ABB RobotStudio station: Assignment2_task#2_20200910-153317.rsstn

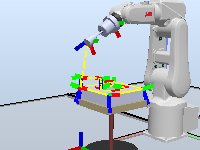
Station Assignment2_task#2 (saved by RobotStudio 20.1.9014.1)
Controller Controller3, task T_ROB1: task frame (RAPID world) sits at (100, 100, 0) mm in the station
Controller Controller3
  mechanical unit ROB_1: IRB120_3_58__01, 6 joints, base frame (0, 0, 0) mm
Layout (positions relative to the parent item):
  - IRB120_3_58__01 [mechanism, from Robots\IRB120_3_58_G_01.rslib] at (100, 100, 0) mm; joint values [0, 0, 0, 0, 0.5236, 0] (rad or m)
  - AssemblySpindleSide [part] at (447.83, 171.64, 630.14) mm, rotated rx -90 ry 60 rz 180 deg
  - Task2_Part [part] at (570, 0, 250) mm, rotated rx 90 ry 0 rz 90 deg
  - Table [part] at (15, -15, 220) mm
  - LegBase [part] at (-100, 100, 0) mm
  - LegSupport [part] at (-100, 100, 0) mm
Attachment: AssemblySpindleSide is attached to IRB120_3_58__01 / Link6
Attachment: LegSupport is attached to Table
Attachment: LegBase is attached to LegSupport
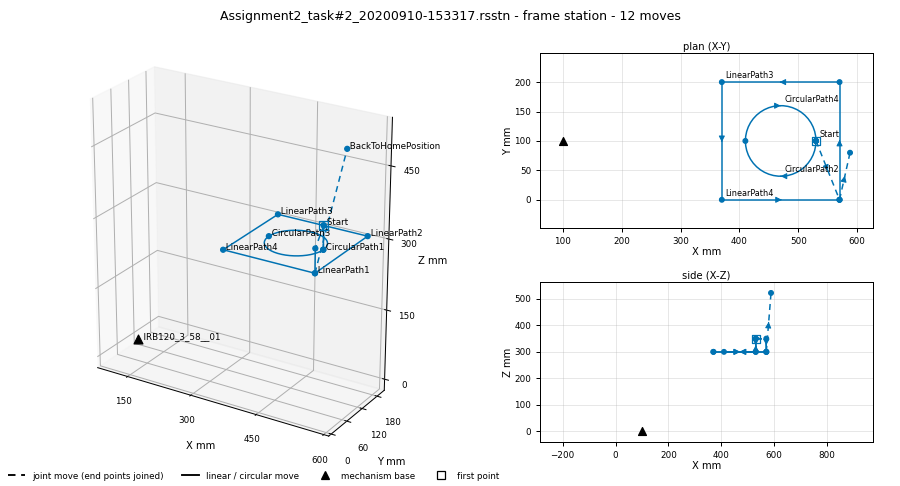
[picture p0: tool path of Assignment2_task#2_20200910-153317.rsstn in frame station, 12 of 12 moves have a stored position in this frame; points joined in program order, loops and branches not executed]
Targets, tools, work objects and paths stored in the station, written as RAPID:
! task T_ROB1
MODULE CalibData
  TASK PERS tooldata Tooldata_1:=[TRUE,[[0,-20.001,142.61],[1,0,0,0]],[1,[0,0,1],[1,0,0,0],0,0,0]];
  TASK PERS wobjdata task2:=[FALSE,TRUE,"",[[470,-100,0],[0.707106781,0,0,0.707106781]],[[0,0,0],[1,0,0,0]]];
  TASK PERS wobjdata LegBase:=[FALSE,TRUE,"",[[470,-100,10],[1,0,0,0]],[[0,0,0],[1,0,0,0]]];
ENDMODULE

! task T_ROB1
MODULE Module1
  CONST robtarget CircularPath1:=[[100,40,300],[0,0,0.984807753,0.173648179],[0,0,-1,0],[9E+09,9E+09,9E+09,9E+09,9E+09,9E+09]];
  CONST robtarget CircularPath2:=[[40,100,300],[0.122787804,0.69636424,0.69636424,0.122787804],[-1,0,-1,0],[9E+09,9E+09,9E+09,9E+09,9E+09,9E+09]];
  CONST robtarget CircularPath3:=[[100,160,300],[0.130526193,0.991444861,0,0],[0,0,0,0],[9E+09,9E+09,9E+09,9E+09,9E+09,9E+09]];
  CONST robtarget CircularPath4:=[[160,100,300],[0.122787804,0.69636424,-0.69636424,-0.122787804],[0,-1,2,0],[9E+09,9E+09,9E+09,9E+09,9E+09,9E+09]];
  CONST robtarget CircularPath5:=[[100,40,300],[0,0,0.984807753,0.173648178],[0,-1,2,0],[9E+09,9E+09,9E+09,9E+09,9E+09,9E+09]];
  CONST robtarget Start:=[[100,40,350],[0,0,1,0],[0,0,-1,0],[9E+09,9E+09,9E+09,9E+09,9E+09,9E+09]];
  CONST robtarget lift:=[[100,40,350],[0,0,1,0],[0,0,3,0],[9E+09,9E+09,9E+09,9E+09,9E+09,9E+09]];
  CONST robtarget Start2:=[[0,0,350],[0,1,0,0],[-1,0,0,0],[9E+09,9E+09,9E+09,9E+09,9E+09,9E+09]];
  CONST robtarget Lift2:=[[0,0,350],[0,-0.707106781,0.707106781,0],[-1,0,-3,0],[9E+09,9E+09,9E+09,9E+09,9E+09,9E+09]];
  CONST robtarget BackToHomePosition:=[[17.857711906,79.999,512.695],[0.5,0,0.866025404,0],[0,0,0,0],[9E+09,9E+09,9E+09,9E+09,9E+09,9E+09]];
  CONST robtarget LinearPath1:=[[0,0,290],[0.092295956,0.701057385,0.701057385,0.092295956],[0,0,0,0],[9E+09,9E+09,9E+09,9E+09,9E+09,9E+09]];
  CONST robtarget LinearPath2:=[[0,200,290],[0.037584344,0.213151409,0.961463877,0.169532023],[0,0,1,0],[9E+09,9E+09,9E+09,9E+09,9E+09,9E+09]];
  CONST robtarget LinearPath3:=[[-200,200,290],[0.073386891,0.416197739,-0.892538936,-0.157378695],[0,0,0,0],[9E+09,9E+09,9E+09,9E+09,9E+09,9E+09]];
  CONST robtarget LinearPath4:=[[-200,0,290],[0.163175911,0.925416578,-0.336824089,-0.059391175],[-1,0,-2,0],[9E+09,9E+09,9E+09,9E+09,9E+09,9E+09]];
  CONST robtarget LinearPath5:=[[0,0,290],[0.160429998,0.909843727,0.376869609,0.06645228],[-1,0,-3,0],[9E+09,9E+09,9E+09,9E+09,9E+09,9E+09]];
  PROC Path_10()
    MoveJ Start,v100,z10,Tooldata_1\WObj:=task2;
    MoveL CircularPath1,v100,z10,Tooldata_1\WObj:=task2;
    MoveC CircularPath2,CircularPath3,v100,z10,Tooldata_1\WObj:=task2;
    MoveC CircularPath4,CircularPath5,v100,z10,Tooldata_1\WObj:=task2;
    MoveJ lift,v100,z10,Tooldata_1\WObj:=task2;
    MoveJ Start2,v100,z10,Tooldata_1\WObj:=task2;
    MoveL LinearPath1,v100,z10,Tooldata_1\WObj:=LegBase;
    MoveL LinearPath2,v100,z10,Tooldata_1\WObj:=LegBase;
    MoveL LinearPath3,v100,z10,Tooldata_1\WObj:=LegBase;
    MoveL LinearPath4,v100,z10,Tooldata_1\WObj:=LegBase;
    MoveL LinearPath5,v100,z10,Tooldata_1\WObj:=LegBase;
    MoveJ BackToHomePosition,v100,z10,Tooldata_1\WObj:=LegBase;
  ENDPROC
  PROC main()
    Path_10;
  ENDPROC
ENDMODULE

